// TIA Portal project "mophongban2" (V20)

(* hardware
DEVICE "S7-1500/ET200MP station_1"  S7-1500 station
   slot 0: "Rail_0"  Rack  6ES7 590-1***0-0AA0
   slot 1: "PLC_1"  CPU 1516-3 PN/DP  6ES7 516-3AP03-0AB0  V4.0
      slot 3: "CPU display_1"  6ES7591-1BA00-0AA0
      slot 32768: "PROFINET interface_1"  X1
         slot 32769: "Port_1"  X1 P1
         slot 32770: "Port_2"  X1 P2
      slot 33024: "PROFINET interface_2"  X2
         slot 33025: "Port_1"  X2 P1
      slot 33280: "DP interface_1"  X3
      slot 34817: "Virtual CP interface port_1"  Virtual CP interface port  Virtual CP interface port FW V4.0
*)

// ===== PLC "PLC_1"  CPU 1516-3 PN/DP =====

DATA_BLOCK "DB_VFD_Fault"   // DB1
{ S7_Optimized_Access := 'FALSE' }
VERSION : 0.1
// QUAN TRONG: DB nay PHAI o che do "Standard - compatible" (khong toi uu hoa).
//  Sau khi Generate blocks from source, mo DB > chuot phai > Properties > Attributes
//  > bo tick "Optimized block access". Neu con optimized, python-snap7 doc offset
//  se ra sai gia tri ma KHONG bao loi (loi kho phat hien nhat).
// 
//  Chi con 2 nut mo phong loi: lá»—i dÃ²ng (Overcurrent) va lá»—i nhiá»‡t (Overtemperature) -
//  moi nut chi lam tang dung 1 gia tri tuong ung (Current_A hoac Temperature_C).
// 
//  Thu tu bien duoc thiet ke co y de offset de doan (xem docs-thiet-ke/Worksheet-Thiet-Ke-DB-Mo-Phong.md):
//    Byte 0, bit 0 : SimButton_OverCurrent      (nut loi dong)
//    Byte 0, bit 1 : FaultActive
//    Byte 0, bit 2 : ResetFault
//    Byte 0, bit 3 : SimButton_Overtemperature  (nut loi nhiet)
//    Byte 0, bit 4 : CurrentFaultLatched        (noi bo FB - dang loi dong)
//    Byte 0, bit 5 : TemperatureFaultLatched    (noi bo FB - dang loi nhiet)
//    Byte 2        : FaultCode   (Int can byte chan, TIA se tu chen padding byte 1)
//    Byte 4        : FaultEventID (Int)
//    Byte 6, bit 0 : SystemOn (Int/Real can byte chan, TIA se tu chen padding con lai cua byte 6-7)
//    Byte 8        : Current_A (Real)
//    Byte 12       : Temperature_C (Real)
//  Sau khi Generate blocks from source, BAT BUOC mo view "Extended" trong TIA de
//  xac nhan lai offset that roi doi tuong ung trong python-bridge/.env neu khac.
   VAR
      SimButton_OverCurrent : Bool;   // Nut nhan mo phong loi dong (Overcurrent) - ep TRUE qua Watch Table (giu >=1 chu ky quet roi tha ve FALSE)
      FaultActive : Bool;   // TRUE = dang co loi (latch boi FB_SimulateVFDFault) - python-bridge doc bit nay
      ResetFault : Bool;   // Ghi TRUE (tu Watch Table hoac python-bridge) de xoa loi - FB tu dua ve FALSE sau 1 chu ky
      SimButton_Overtemperature : Bool;   // Nut nhan mo phong loi nhiet (Overtemperature) - ep TRUE qua Watch Table (giu >=1 chu ky quet roi tha ve FALSE)
      CurrentFaultLatched : Bool;   // Noi bo (FB dung): TRUE khi loi dang active la loi dong - dieu khien Current_A
      TemperatureFaultLatched : Bool;   // Noi bo (FB dung): TRUE khi loi dang active la loi nhiet - dieu khien Temperature_C
      FaultCode : Int;   // 0 = khong loi, 1 = loi dong, 2 = loi nhiet - xem python-bridge/data/fault_codes_v20.json
      FaultEventID : Int;   // Tang dan moi lan co loi MOI (canh len cua bat ky SimButton nao) - python-bridge dung de tranh gui trung lap
      SystemOn : Bool;   // Nut ON/OFF he thong - TRUE = dang chay, mo phong dong dien/nhiet do binh thuong
      Current_A : Real;   // Dong dien mo phong (A) - binh thuong 8.0, tang len 8.5 (vua vuot nguong) khi loi dong dang active
      Temperature_C : Real;   // Nhiet do mo phong (do C) - binh thuong 50.0, tang len 95.0 khi loi nhiet dang active
   END_VAR
BEGIN
END_DATA_BLOCK

DATA_BLOCK "FB_SimulateVFDFault_DB"   // DB2
{ S7_Optimized_Access := 'TRUE' }
VERSION : 0.5
// stored: InstanceOfName FB_SimulateVFDFault
"FB_SimulateVFDFault"
BEGIN
END_DATA_BLOCK

DATA_BLOCK "FB_SimulateVFDFault_DB_1"   // DB3
{ S7_Optimized_Access := 'TRUE' }
VERSION : 0.6
// stored: InstanceOfName FB_SimulateVFDFault
"FB_SimulateVFDFault"
BEGIN
END_DATA_BLOCK

DATA_BLOCK "FB_SimulateVFDFault_DB_2"   // DB4
{ S7_Optimized_Access := 'TRUE' }
VERSION : 0.7
// stored: InstanceOfName FB_SimulateVFDFault
"FB_SimulateVFDFault"
BEGIN
END_DATA_BLOCK

FUNCTION_BLOCK "FB_SimulateVFDFault"   // FB1, SCL
{ S7_Optimized_Access := 'TRUE' }
VERSION : 0.7
// Goi khoi nay moi chu ky quet trong OB1 (Main), khong can tham so IN/OUT -
//  doc/ghi truc tiep "DB_VFD_Fault" vi day chi la logic mo phong don gian cho do an.
//  Tao 1 Instance DB rieng khi keo vao OB1 (vi du "IDB_SimulateVFDFault").
// 
//  Chi con 2 nut loi doc lap voi nhau, CHI CO TAC DUNG KHI SystemOn = TRUE
//  (may chua bat thi khong the "qua dong"/"qua nhiet"):
//    - SimButton_OverCurrent     (nut loi dong)  -> chi day Current_A len, khong dung Temperature_C
//    - SimButton_Overtemperature (nut loi nhiet)  -> chi day Temperature_C len, khong dung Current_A
// 
//  Current_A/Temperature_C KHONG con nhay tuc thi - moi RAMP_STEP_TIME (500ms)
//  tang/giam dan 1 buoc (CURRENT_STEP/TEMPERATURE_STEP):
//    - SystemOn = FALSE                -> giam dan ve 0.0 (may tat)
//    - SystemOn = TRUE, khong co loi   -> tien ve gia tri binh thuong (Current_A=8.0, Temperature_C=50.0), tu duoi len hoac tu tren xuong (vd sau khi Reset)
//    - SystemOn = TRUE, loi dang active-> TANG LIEN TUC KHONG GIOI HAN (khong co tran) cho toi khi ResetFault
//  Tat SystemOn (OFF) hoac ResetFault se xoa loi dang active (FaultActive/FaultCode ve 0,
//  gia tri tu dong giam dan ve lai binh thuong/0 theo nhanh tren).
   VAR
      risingEdgeButton : R_TRIG;   // Nut loi dong (Overcurrent)
      risingEdgeOvertemperature : R_TRIG;   // Nut loi nhiet (Overtemperature)
      rampTimer : TON_TIME;   // Tao xung dieu khien moi RAMP_STEP_TIME
      rampPulse : Bool;   // Bien trung gian giu Q chu ky truoc - tranh tu tham chieu #rampTimer.Q lam IN cho chinh no
      CURRENT_NORMAL : Real := 8.0;   // Dong dien binh thuong (A)
      TEMPERATURE_NORMAL : Real := 50.0;   // Nhiet do binh thuong (do C)
      CURRENT_STEP : Real := 0.5;   // Dong dien tang/giam moi buoc (A)
      TEMPERATURE_STEP : Real := 1.5;   // Nhiet do tang/giam moi buoc (do C)
      RAMP_STEP_TIME : Time := T#500MS;   // Chu ky 1 buoc tang/giam
   END_VAR
BEGIN

   // Nhan nut mo phong loi dong -> chi tinh khi SystemOn=TRUE (may dang chay)
   #risingEdgeButton(CLK := "DB_VFD_Fault".SimButton_OverCurrent);
   IF #risingEdgeButton.Q AND "DB_VFD_Fault".SystemOn THEN
       "DB_VFD_Fault".FaultActive := TRUE;
       "DB_VFD_Fault".FaultCode := 1; // 1 = Loi dong (Overcurrent) - xem fault_codes_v20.json
       "DB_VFD_Fault".FaultEventID := "DB_VFD_Fault".FaultEventID + 1;
       "DB_VFD_Fault".CurrentFaultLatched := TRUE;
       "DB_VFD_Fault".TemperatureFaultLatched := FALSE;
   END_IF;

   // Nhan nut mo phong loi nhiet -> chi tinh khi SystemOn=TRUE (may dang chay)
   #risingEdgeOvertemperature(CLK := "DB_VFD_Fault".SimButton_Overtemperature);
   IF #risingEdgeOvertemperature.Q AND "DB_VFD_Fault".SystemOn THEN
       "DB_VFD_Fault".FaultActive := TRUE;
       "DB_VFD_Fault".FaultCode := 2; // 2 = Loi nhiet (Overtemperature) - xem fault_codes_v20.json
       "DB_VFD_Fault".FaultEventID := "DB_VFD_Fault".FaultEventID + 1;
       "DB_VFD_Fault".TemperatureFaultLatched := TRUE;
       "DB_VFD_Fault".CurrentFaultLatched := FALSE;
   END_IF;

   // Xoa loi: Watch Table hoac python-bridge ghi ResetFault := TRUE - cung tha
   // luon 2 nut loi ve FALSE (phong truong hop ep qua Watch Table quen tha nut)
   IF "DB_VFD_Fault".ResetFault THEN
       "DB_VFD_Fault".FaultActive := FALSE;
       "DB_VFD_Fault".FaultCode := 0;
       "DB_VFD_Fault".CurrentFaultLatched := FALSE;
       "DB_VFD_Fault".TemperatureFaultLatched := FALSE;
       "DB_VFD_Fault".SimButton_OverCurrent := FALSE;
       "DB_VFD_Fault".SimButton_Overtemperature := FALSE;
       "DB_VFD_Fault".ResetFault := FALSE;
   END_IF;

   // Tat he thong thi tu dong xoa loi luon (khong the "dang loi" khi may da tat)
   IF NOT "DB_VFD_Fault".SystemOn THEN
       "DB_VFD_Fault".FaultActive := FALSE;
       "DB_VFD_Fault".FaultCode := 0;
       "DB_VFD_Fault".CurrentFaultLatched := FALSE;
       "DB_VFD_Fault".TemperatureFaultLatched := FALSE;
   END_IF;

   // Timer tu dao (self-retrigger) qua bien trung gian rampPulse - KHONG doc truc
   // tiep #rampTimer.Q lam IN cho chinh no (mot so ban SCL xu ly tu tham chieu
   // nay khong on dinh, khien Q khong bao gio thuc su len TRUE).
   #rampTimer(IN := NOT #rampPulse,
              PT := #RAMP_STEP_TIME);
   #rampPulse := #rampTimer.Q;
   IF #rampTimer.Q THEN
       // ----- Dong dien -----
       IF NOT "DB_VFD_Fault".SystemOn THEN
           // May tat: giam dan ve 0.0
           IF "DB_VFD_Fault".Current_A > 0.0 THEN
               "DB_VFD_Fault".Current_A := "DB_VFD_Fault".Current_A - #CURRENT_STEP;
               IF "DB_VFD_Fault".Current_A < 0.0 THEN
                   "DB_VFD_Fault".Current_A := 0.0;
               END_IF;
           END_IF;
       ELSIF "DB_VFD_Fault".CurrentFaultLatched THEN
           // Dang loi dong: tang lien tuc, KHONG gioi han tran
           "DB_VFD_Fault".Current_A := "DB_VFD_Fault".Current_A + #CURRENT_STEP;
       ELSE
           // Binh thuong: tien ve CURRENT_NORMAL (8.0) - tu duoi len (moi bat may)
           // hoac tu tren xuong (vua Reset sau khi loi tang cao)
           IF "DB_VFD_Fault".Current_A < #CURRENT_NORMAL THEN
               "DB_VFD_Fault".Current_A := "DB_VFD_Fault".Current_A + #CURRENT_STEP;
               IF "DB_VFD_Fault".Current_A > #CURRENT_NORMAL THEN
                   "DB_VFD_Fault".Current_A := #CURRENT_NORMAL;
               END_IF;
           ELSIF "DB_VFD_Fault".Current_A > #CURRENT_NORMAL THEN
               "DB_VFD_Fault".Current_A := "DB_VFD_Fault".Current_A - #CURRENT_STEP;
               IF "DB_VFD_Fault".Current_A < #CURRENT_NORMAL THEN
                   "DB_VFD_Fault".Current_A := #CURRENT_NORMAL;
               END_IF;
           END_IF;
       END_IF;

       // ----- Nhiet do ----- (tuong tu dong dien, muc binh thuong 50.0)
       IF NOT "DB_VFD_Fault".SystemOn THEN
           IF "DB_VFD_Fault".Temperature_C > 0.0 THEN
               "DB_VFD_Fault".Temperature_C := "DB_VFD_Fault".Temperature_C - #TEMPERATURE_STEP;
               IF "DB_VFD_Fault".Temperature_C < 0.0 THEN
                   "DB_VFD_Fault".Temperature_C := 0.0;
               END_IF;
           END_IF;
       ELSIF "DB_VFD_Fault".TemperatureFaultLatched THEN
           // Dang loi nhiet: tang lien tuc, KHONG gioi han tran
           "DB_VFD_Fault".Temperature_C := "DB_VFD_Fault".Temperature_C + #TEMPERATURE_STEP;
       ELSE
           IF "DB_VFD_Fault".Temperature_C < #TEMPERATURE_NORMAL THEN
               "DB_VFD_Fault".Temperature_C := "DB_VFD_Fault".Temperature_C + #TEMPERATURE_STEP;
               IF "DB_VFD_Fault".Temperature_C > #TEMPERATURE_NORMAL THEN
                   "DB_VFD_Fault".Temperature_C := #TEMPERATURE_NORMAL;
               END_IF;
           ELSIF "DB_VFD_Fault".Temperature_C > #TEMPERATURE_NORMAL THEN
               "DB_VFD_Fault".Temperature_C := "DB_VFD_Fault".Temperature_C - #TEMPERATURE_STEP;
               IF "DB_VFD_Fault".Temperature_C < #TEMPERATURE_NORMAL THEN
                   "DB_VFD_Fault".Temperature_C := #TEMPERATURE_NORMAL;
               END_IF;
           END_IF;
       END_IF;
   END_IF;
END_FUNCTION_BLOCK

ORGANIZATION_BLOCK "Main"   // OB1, LAD, ProgramCycle
TITLE = "Main Program Sweep (Cycle)"
{ S7_Optimized_Access := 'TRUE' }
VERSION : 0.1
   VAR_INPUT
      Initial_Call : Bool;   // Initial call of this OB
      Remanence : Bool;   // =True, if remanent data are available
   END_VAR
BEGIN

REGION Network 1
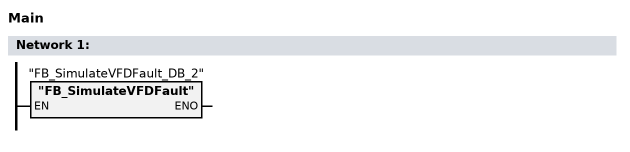
   RUNG wire#powerrail
      "FB_SimulateVFDFault_DB_2"()
   END_RUNG
   // the same network as SCL:
   "FB_SimulateVFDFault_DB_2"();   // "FB_SimulateVFDFault"
END_REGION
END_ORGANIZATION_BLOCK